Fanuc KAREL source: CNV_STR_INT.kl

PROGRAM T
%NOLOCKGROUP
VAR
 v0 : STRING[40]
 v1 : INTEGER
BEGIN
 CNV_STR_INT(v0, v1)
END T
